TYPE OutputBase_10CEE7DE :
STRUCT
END_STRUCT
END_TYPE

(* stored: Version 1.1.0.1, ProductVersion 3.1.4024.9
   DUT OutputBase_10CEE7DE: Id {1e1c7eed-151b-42f1-a168-0e08fe624324} *)
